FUNCTION F_Byte_To_Word : WORD
VAR_INPUT
	bByte0	: BYTE;
	bByte1	: BYTE;
END_VAR
VAR
END_VAR

MEMCPY(ADR(F_Byte_To_Word),ADR(bByte0),SIZEOF(bByte0)); (*set  zero*)
MEMCPY(ADR(F_Byte_To_Word)+1,ADR(bByte1),SIZEOF(bByte0)); (*set  zero*)

END_FUNCTION

(* stored: Version 1.1.0.1, ProductVersion 3.1.4024.11
   POU F_Byte_To_Word: Id {5531a254-d487-412b-8d10-ceba450657f9}, SpecialFunc None *)
